FUNCTION_BLOCK FB_SL3K4ReadPMPSDB
VAR_INPUT
    sDeviceName      : STRING;
    bFileReaderBusy  : BOOL;
    bFileReaderError : BOOL;
    sTransitionKey   : STRING;
    jsonDoc          : SJsonValue;
END_VAR

VAR_IN_OUT
    fbFFHWO          : FB_HardwareFFOutput;	
END_VAR

VAR
    fbJsonLoader: FB_JsonDocToSafeBP;
    ffError     : FB_FastFault;
    ftDbBusy    : F_TRIG;
    ftRead      : F_TRIG;
    bReadPmpsDb : BOOL := FALSE;
    i           : INT;
END_VAR

VAR_OUTPUT
    astDbStateParams   : ARRAY[0..GeneralConstants.MAX_STATES] OF ST_DbStateParams;
    bLoadedNormal      : BOOL;
    bLoadedMaintenance : BOOL;
    bFirstReadDone     : BOOL;
    bError             : BOOL;
    bStatesReady       : BOOL;
    bAllStatesLoaded   : BOOL;
    nErrId             : UDINT;
    sErrMsg            : STRING;
END_VAR

// Only reload and assert if external fast fault output is valid
IF NOT __ISVALIDREF(fbFFHWO) THEN
    RETURN;
END_IF

// Map state strings for DB lookup (indexing strictly controlled/setup by config/tool)
astDbStateParams[0].sPmpsState := sTransitionKey; // Transition state
astDbStateParams[1].sPmpsState := 'NORMAL';
astDbStateParams[2].sPmpsState := 'MAINTENANCE';

// --- Edge-trigger: Only reload DB when reader finishes (Busy->not busy)
ftDbBusy(CLK := bFileReaderBusy);
IF ftDbBusy.Q THEN
    bReadPmpsDb := NOT bFileReaderError; // One-shot trigger: only reload if successful parse
END_IF

// Call JSON loader to parse PMPS parameters
fbJsonLoader(
    bExecute    := bReadPmpsDb,
    jsonDoc     := jsonDoc,
    sDeviceName := sDeviceName,
    arrStates   := astDbStateParams,
    io_fbFFHWO  := fbFFHWO
);
// Reset reload request when JSON loader is done (not busy)
IF NOT fbJsonLoader.bBusy THEN
    bReadPmpsDb := FALSE;
END_IF

// Track first DB read completion
ftRead(CLK := fbJsonLoader.bBusy);
IF ftRead.Q AND NOT fbJsonLoader.bError THEN
    bFirstReadDone := TRUE;
END_IF

// Error outputs and reporting
bError  := fbJsonLoader.bError;
nErrId  := fbJsonLoader.nErrId;
sErrMsg := fbJsonLoader.sErrMsg;

// --- Check if all state params are loaded (including transition, normal, maintenance) ---
bAllStatesLoaded := TRUE;
FOR i := 0 TO 2 DO
    bAllStatesLoaded := bAllStatesLoaded AND astDbStateParams[i].bBeamParamsLoaded;
END_FOR

bLoadedNormal      := astDbStateParams[1].bBeamParamsLoaded;
bLoadedMaintenance := astDbStateParams[2].bBeamParamsLoaded;

// Final readiness: device is ready only when DB load finished successfully and all states loaded
bStatesReady := (fbJsonLoader.bBusy = FALSE) AND (NOT bError) AND bAllStatesLoaded;

// Fast fault handling for loader or DB error
ffError(
    i_xOK        := NOT bError,
    i_xAutoReset := TRUE,
    i_DevName    := sDeviceName,
    i_Desc       := 'PMPS DB load error (TRANSITION/NORMAL/MAINTENANCE)',
    i_TypeCode   := E_MotionFFType.INTERNAL_ERROR,
    io_fbFFHWO   := fbFFHWO
);

END_FUNCTION_BLOCK

(* stored: Version 1.1.0.1
   POU FB_SL3K4ReadPMPSDB: Id {bbf2cac6-9f54-4c2d-b415-c76e1add5790}, SpecialFunc None *)
